// TIA Portal V16 export
// export: Created 2022-09-01T14:29:20.9311088Z, ExportSetting WithDefaults, DisplayName Totally Integrated Automation Portal, DisplayVersion V16, DisplayName TIA Portal Version Control Interface, DisplayVersion V16, DisplayName TIA Portal Openness, DisplayVersion V16, DisplayName STEP 7 Professional, DisplayVersion V16, DisplayName STEP 7 Safety, DisplayVersion V16, DisplayName WinCC Advanced, DisplayVersion V16
FUNCTION "Reset_Etapas_Iniciais" : Void   // FC23, LAD
TITLE = Reset às etapas inicias em caso de falha de energia, de modo e continuar o processo do ponto onde estava
{ S7_Optimized_Access := 'TRUE' }
VERSION : 0.1
// stored: AutoNumber true, IsIECCheckEnabled false, SetENOAutomatically false, UDAEnableTagReadback false
BEGIN

REGION Network 1: Reset etapa 1
   // as etapas 3, 33 e 7 não precisam nem devem fazer reset à etapa 1. Já é feito indiretamente no FC4
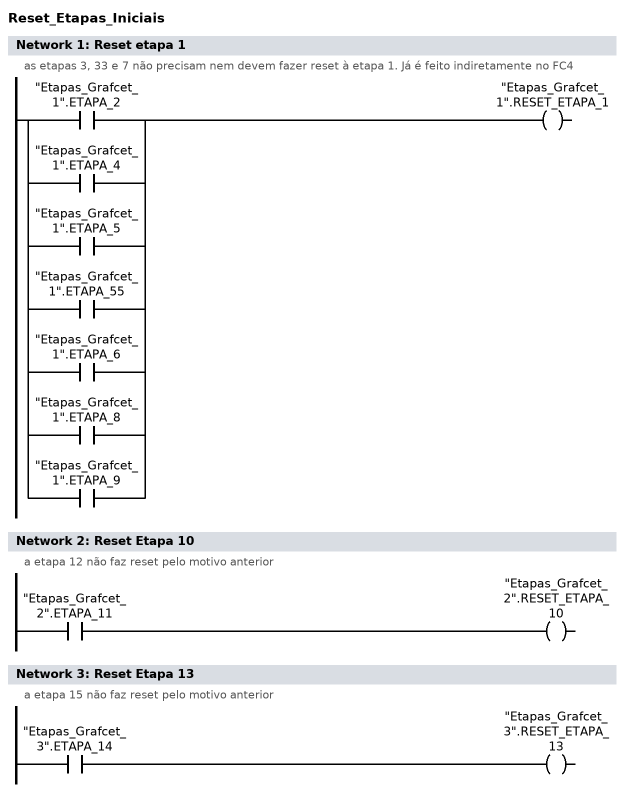
   RUNG wire#powerrail
      Contact( "Etapas_Grafcet_1".ETAPA_2 )
      wire#w1
      Coil( "Etapas_Grafcet_1".RESET_ETAPA_1 )
   END_RUNG
   RUNG wire#powerrail
      Contact( "Etapas_Grafcet_1".ETAPA_4 )
   END_RUNG wire#w1
   RUNG wire#powerrail
      Contact( "Etapas_Grafcet_1".ETAPA_5 )
   END_RUNG wire#w1
   RUNG wire#powerrail
      Contact( "Etapas_Grafcet_1".ETAPA_55 )
   END_RUNG wire#w1
   RUNG wire#powerrail
      Contact( "Etapas_Grafcet_1".ETAPA_6 )
   END_RUNG wire#w1
   RUNG wire#powerrail
      Contact( "Etapas_Grafcet_1".ETAPA_8 )
   END_RUNG wire#w1
   RUNG wire#powerrail
      Contact( "Etapas_Grafcet_1".ETAPA_9 )
   END_RUNG wire#w1
   // the same network as SCL:
   "Etapas_Grafcet_1".RESET_ETAPA_1 := "Etapas_Grafcet_1".ETAPA_2 OR "Etapas_Grafcet_1".ETAPA_4 OR "Etapas_Grafcet_1".ETAPA_5 OR "Etapas_Grafcet_1".ETAPA_55 OR "Etapas_Grafcet_1".ETAPA_6 OR "Etapas_Grafcet_1".ETAPA_8 OR "Etapas_Grafcet_1".ETAPA_9;
END_REGION

REGION Network 2: Reset Etapa 10
   // a etapa 12 não faz reset pelo motivo anterior
   RUNG wire#powerrail
      Contact( "Etapas_Grafcet_2".ETAPA_11 )
      Coil( "Etapas_Grafcet_2".RESET_ETAPA_10 )
   END_RUNG
   // the same network as SCL:
   "Etapas_Grafcet_2".RESET_ETAPA_10 := "Etapas_Grafcet_2".ETAPA_11;
END_REGION

REGION Network 3: Reset Etapa 13
   // a etapa 15 não faz reset pelo motivo anterior
   RUNG wire#powerrail
      Contact( "Etapas_Grafcet_3".ETAPA_14 )
      Coil( "Etapas_Grafcet_3".RESET_ETAPA_13 )
   END_RUNG
   // the same network as SCL:
   "Etapas_Grafcet_3".RESET_ETAPA_13 := "Etapas_Grafcet_3".ETAPA_14;
END_REGION
END_FUNCTION
